ADAPTER EventAdapter
  (* Standard: 61499-1 *)
  (* Version 1.0, 2023-03-07, AK115394 *)
  (* Compiler header: package fb.test; *)
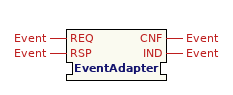
  EVENT_INPUT
    REQ;
    RSP;
  END_EVENT
  EVENT_OUTPUT
    CNF;
    IND;
  END_EVENT
  SERVICE PLUG/SOCKET
    SEQUENCE request_confirm
      SOCKET.REQ(REQD) -> PLUG.REQ(REQD);
      PLUG.CNF(CNFD) -> SOCKET.CNF(CNFD);
    END_SEQUENCE
    SEQUENCE indication_response
      PLUG.IND(INDD) -> SOCKET.IND(INDD);
      SOCKET.RSP(RSPD) -> PLUG.RSP(RSPD);
    END_SEQUENCE
  END_SERVICE
END_ADAPTER
